// Mitsubishi GX Works2 project: Ex01   PLC: Q02/Q02H

PROGRAM MAIN
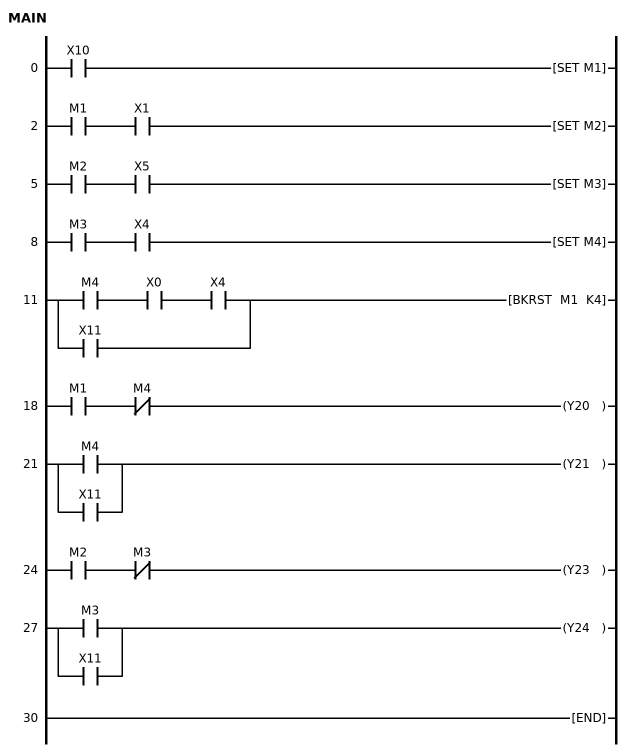
0     LD      X10
      SET     M1
2     LD      M1
      AND     X1
      SET     M2
5     LD      M2
      AND     X5
      SET     M3
8     LD      M3
      AND     X4
      SET     M4
11    LD      M4
      AND     X0
      AND     X4
      OR      X11
      BKRST   M1 K4
18    LD      M1
      ANI     M4
      OUT     Y20
21    LD      M4
      OR      X11
      OUT     Y21
24    LD      M2
      ANI     M3
      OUT     Y23
27    LD      M3
      OR      X11
      OUT     Y24
30    END
END_PROGRAM
